FUNCTION_BLOCK Pass10
  (* Standard: 61499-2 *)
  (* Version 0.1, 2017-00-01, hpea485, UOA *)
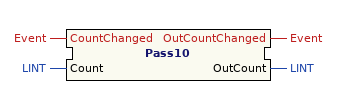
  EVENT_INPUT
    CountChanged;
  END_EVENT
  EVENT_OUTPUT
    OutCountChanged;
  END_EVENT
  VAR_INPUT
    Count : LINT;
  END_VAR
  VAR_OUTPUT
    OutCount : LINT;
  END_VAR
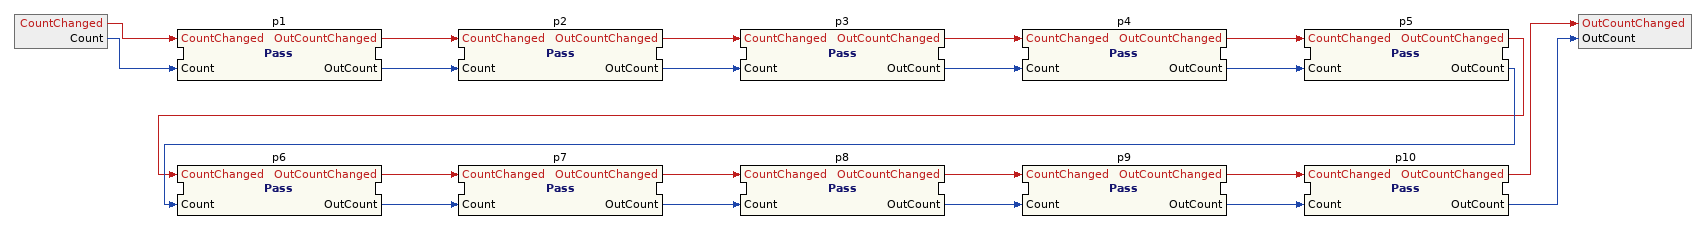
  FBS
    p1 : Pass;
    p2 : Pass;
    p3 : Pass;
    p4 : Pass;
    p5 : Pass;
    p9 : Pass;
    p6 : Pass;
    p10 : Pass;
    p7 : Pass;
    p8 : Pass;
  END_FBS
  EVENT_CONNECTIONS
    CountChanged TO p1.CountChanged;
    p10.OutCountChanged TO OutCountChanged;
    p1.OutCountChanged TO p2.CountChanged;
    p2.OutCountChanged TO p3.CountChanged;
    p3.OutCountChanged TO p4.CountChanged;
    p4.OutCountChanged TO p5.CountChanged;
    p5.OutCountChanged TO p6.CountChanged;
    p9.OutCountChanged TO p10.CountChanged;
    p6.OutCountChanged TO p7.CountChanged;
    p7.OutCountChanged TO p8.CountChanged;
    p8.OutCountChanged TO p9.CountChanged;
  END_CONNECTIONS
  DATA_CONNECTIONS
    Count TO p1.Count;
    p10.OutCount TO OutCount;
    p1.OutCount TO p2.Count;
    p2.OutCount TO p3.Count;
    p3.OutCount TO p4.Count;
    p4.OutCount TO p5.Count;
    p5.OutCount TO p6.Count;
    p9.OutCount TO p10.Count;
    p6.OutCount TO p7.Count;
    p7.OutCount TO p8.Count;
    p8.OutCount TO p9.Count;
  END_CONNECTIONS
END_FUNCTION_BLOCK
